FUNCTION_BLOCK IN_MATRIX (* MATRIX input from table *)
  (* Standard: 61499-2 *)
  (* Version 0.4, 2007-12-17, JHC, Holobloc Inc., Updated IVAL comment. *)
  (* Version 0.3, 2007-10-19, JHC, Holobloc Inc., Moved to fb.rt.hmi.matrix. *)
  (* Version 0.2, 2007-03-15, JHC, Holobloc Inc., Updated IVAL documentation. *)
  (* Version 0.1, 2006-03-19, JHC, Holobloc Inc., Changed package to fb.rt.hmi *)
  (* Version 0.0, 2004-06-22, JHC, Rockwell Automation *)
  (* Compiler header: package fb.rt.hmi.matrix; *)
  (* Compiler classdef: public class IN_MATRIX extends FB_TABLE *)
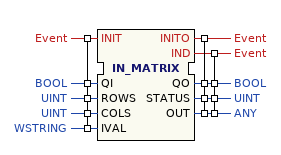
  EVENT_INPUT
    INIT WITH QI, ROWS, COLS, IVAL; (* Initialize matrix to IN *)
  END_EVENT
  EVENT_OUTPUT
    INITO WITH QO, STATUS, OUT; (* Initialization Confirm *)
    IND WITH QO, STATUS, OUT; (* Indication of user input from table *)
  END_EVENT
  VAR_INPUT
    QI : BOOL; (* 1=Enabled,0=Inhibited *)
    ROWS : UINT := 1; (* Number of rows in the table *)
    COLS : UINT := 1; (* Number of columns in the table *)
    IVAL : WSTRING; (* Initial data values, e.g., "[[1,2],[3,4]]" for ROWS=2, COLS=2 *)
  END_VAR
  VAR_OUTPUT
    QO : BOOL; (* 0=OK,1=Inhibited *)
    STATUS : UINT; (* 0=OK,2=TYPE_CONVERSION_ERROR,4=INHIBITED,13=ARRAY_SIZE_ERROR *)
    OUT : ANY; (* Output data from table(implementation-dependent) *)
  END_VAR
END_FUNCTION_BLOCK
